(* Logix 5000 project; controller VET 1756-L62 rev 19.52; software revision 19.01; part 27 of 27 *)
(* tags used below, declared in another part *)
   Aux : DINT[40];
   Color_aux : INT[1000];
   ti : Index;
   _Eqp : Equipo[800];
   _Eqp_Cfg : Eqp_Cfg[800];
   _Origen : Origen[40];
   Set_Global : DINT[20];
(* Typlgie, continued *)

ROUTINE SEQ_MOT_1   (* ladder *)
// Parte 1 se seq. equipos
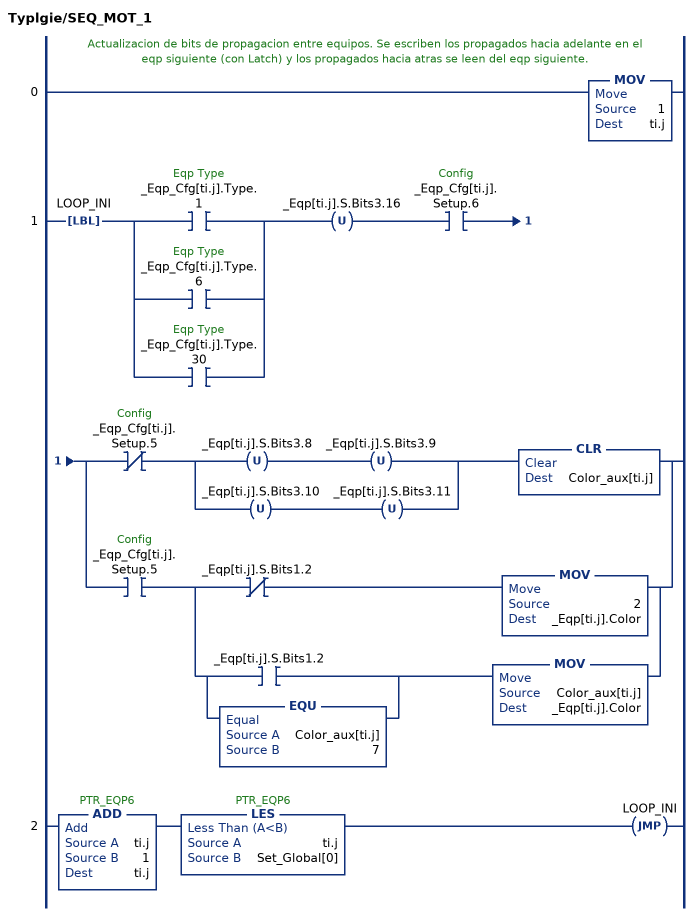
   // Actualizacion de bits de propagacion entre equipos. Se escriben los propagados hacia adelante en el eqp siguiente (con Latch) y los propagados hacia atras se leen del eqp siguiente.
   0: MOV(1,ti.j);
   1: LBL(LOOP_INI)[XIC(_Eqp_Cfg[ti.j].Type.1) ,XIC(_Eqp_Cfg[ti.j].Type.6) ,XIC(_Eqp_Cfg[ti.j].Type.30) ]OTU(_Eqp[ti.j].S.Bits3.16)XIC(_Eqp_Cfg[ti.j].Setup.6)[XIO(_Eqp_Cfg[ti.j].Setup.5) [OTU(_Eqp[ti.j].S.Bits3.8) OTU(_Eqp[ti.j].S.Bits3.9) ,OTU(_Eqp[ti.j].S.Bits3.10) OTU(_Eqp[ti.j].S.Bits3.11) ] CLR(Color_aux[ti.j]) ,XIC(_Eqp_Cfg[ti.j].Setup.5) [XIO(_Eqp[ti.j].S.Bits1.2) MOV(2,_Eqp[ti.j].Color) ,[XIC(_Eqp[ti.j].S.Bits1.2) ,EQU(Color_aux[ti.j],7) ] MOV(Color_aux[ti.j],_Eqp[ti.j].Color) ] ];
   2: ADD(ti.j,1,ti.j)LES(ti.j,Set_Global[0])JMP(LOOP_INI);
END_ROUTINE

ROUTINE SEQ_MOT_2   (* ladder *)
// Parte 2 se seq. equipos
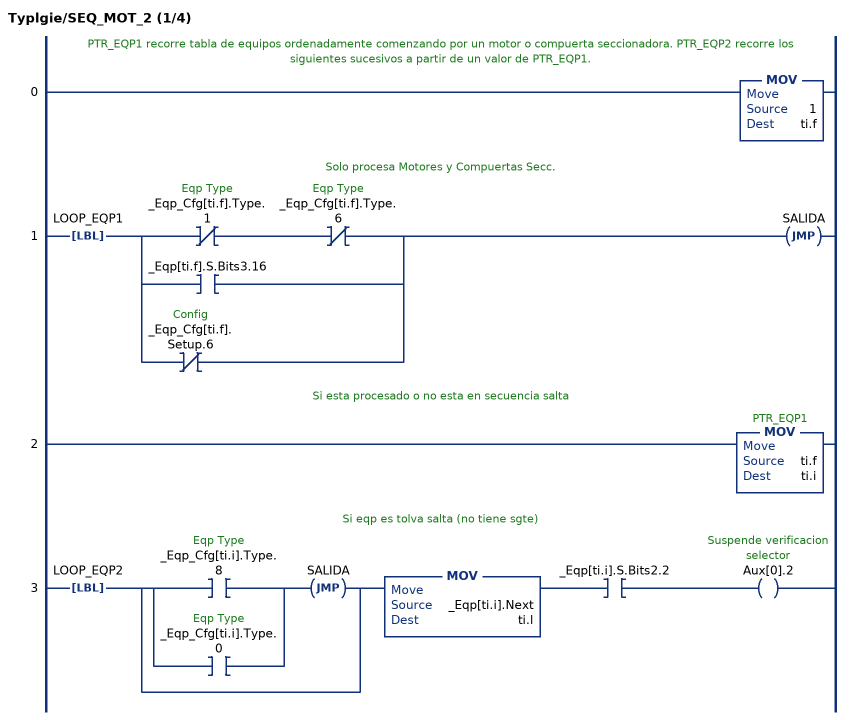
   // PTR_EQP1 recorre tabla de equipos ordenadamente comenzando por un motor o compuerta seccionadora. PTR_EQP2 recorre los siguientes sucesivos a partir de un valor de PTR_EQP1.
   0: MOV(1,ti.f);
   // Solo procesa Motores y Compuertas Secc.
   1: LBL(LOOP_EQP1)[XIO(_Eqp_Cfg[ti.f].Type.1) XIO(_Eqp_Cfg[ti.f].Type.6) ,XIC(_Eqp[ti.f].S.Bits3.16) ,XIO(_Eqp_Cfg[ti.f].Setup.6) ]JMP(SALIDA);
   // Si esta procesado o no esta en secuencia salta
   2: MOV(ti.f,ti.i);
   // Si eqp es tolva salta (no tiene sgte)
   3: LBL(LOOP_EQP2)[[XIC(_Eqp_Cfg[ti.i].Type.8) ,XIC(_Eqp_Cfg[ti.i].Type.0) ] JMP(SALIDA) ,]MOV(_Eqp[ti.i].Next,ti.l)XIC(_Eqp[ti.i].S.Bits2.2)OTE(Aux[0].2);
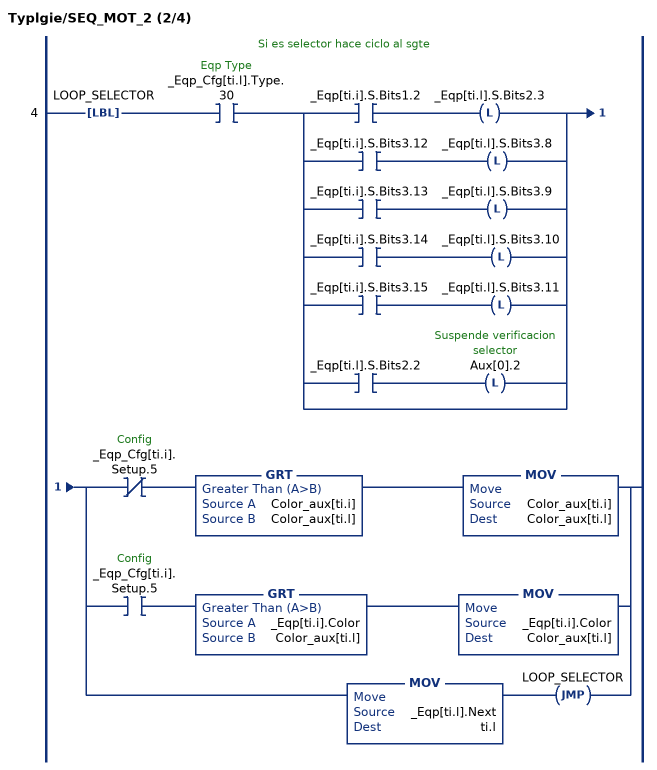
   // Si es selector hace ciclo al sgte
   4: LBL(LOOP_SELECTOR)XIC(_Eqp_Cfg[ti.l].Type.30)[XIC(_Eqp[ti.i].S.Bits1.2) OTL(_Eqp[ti.l].S.Bits2.3) ,XIC(_Eqp[ti.i].S.Bits3.12) OTL(_Eqp[ti.l].S.Bits3.8) ,XIC(_Eqp[ti.i].S.Bits3.13) OTL(_Eqp[ti.l].S.Bits3.9) ,XIC(_Eqp[ti.i].S.Bits3.14) OTL(_Eqp[ti.l].S.Bits3.10) ,XIC(_Eqp[ti.i].S.Bits3.15) OTL(_Eqp[ti.l].S.Bits3.11) ,XIC(_Eqp[ti.l].S.Bits2.2) OTL(Aux[0].2) ,][XIO(_Eqp_Cfg[ti.i].Setup.5) GRT(Color_aux[ti.i],Color_aux[ti.l]) MOV(Color_aux[ti.i],Color_aux[ti.l]) ,XIC(_Eqp_Cfg[ti.i].Setup.5) GRT(_Eqp[ti.i].Color,Color_aux[ti.l]) MOV(_Eqp[ti.i].Color,Color_aux[ti.l]) ,MOV(_Eqp[ti.l].Next,ti.l) JMP(LOOP_SELECTOR) ];
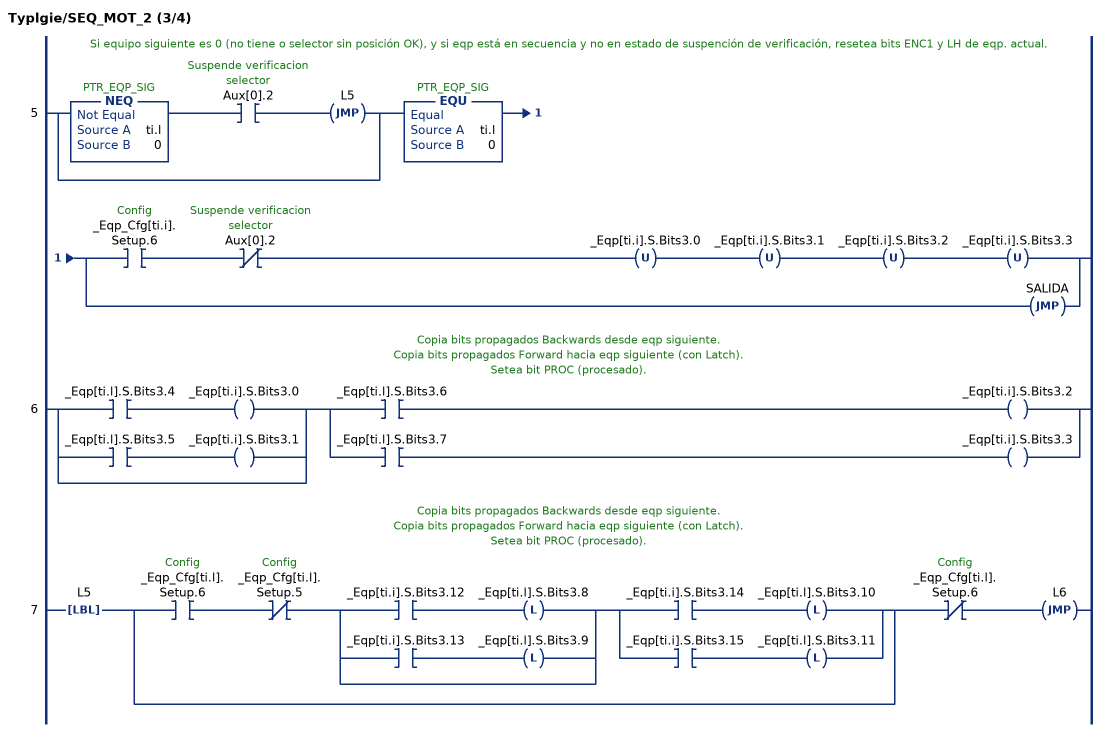
   // Si equipo siguiente es 0 (no tiene o selector sin posición OK), y si eqp está en secuencia y no en estado de suspención de verificación, resetea bits ENC1 y LH de eqp. actual.
   5: [NEQ(ti.l,0) XIC(Aux[0].2) JMP(L5) ,]EQU(ti.l,0)[XIC(_Eqp_Cfg[ti.i].Setup.6) XIO(Aux[0].2) OTU(_Eqp[ti.i].S.Bits3.0) OTU(_Eqp[ti.i].S.Bits3.1) OTU(_Eqp[ti.i].S.Bits3.2) OTU(_Eqp[ti.i].S.Bits3.3) ,JMP(SALIDA) ];
   // Copia bits propagados Backwards desde eqp siguiente.
   // Copia bits propagados Forward hacia eqp siguiente (con Latch).
   // Setea bit PROC (procesado).
   6: [XIC(_Eqp[ti.l].S.Bits3.4) OTE(_Eqp[ti.i].S.Bits3.0) ,XIC(_Eqp[ti.l].S.Bits3.5) OTE(_Eqp[ti.i].S.Bits3.1) ,][XIC(_Eqp[ti.l].S.Bits3.6) OTE(_Eqp[ti.i].S.Bits3.2) ,XIC(_Eqp[ti.l].S.Bits3.7) OTE(_Eqp[ti.i].S.Bits3.3) ];
   // Copia bits propagados Backwards desde eqp siguiente.
   // Copia bits propagados Forward hacia eqp siguiente (con Latch).
   // Setea bit PROC (procesado).
   7: LBL(L5)[XIC(_Eqp_Cfg[ti.l].Setup.6) XIO(_Eqp_Cfg[ti.l].Setup.5) [XIC(_Eqp[ti.i].S.Bits3.12) OTL(_Eqp[ti.l].S.Bits3.8) ,XIC(_Eqp[ti.i].S.Bits3.13) OTL(_Eqp[ti.l].S.Bits3.9) ,] [XIC(_Eqp[ti.i].S.Bits3.14) OTL(_Eqp[ti.l].S.Bits3.10) ,XIC(_Eqp[ti.i].S.Bits3.15) OTL(_Eqp[ti.l].S.Bits3.11) ] ,]XIO(_Eqp_Cfg[ti.l].Setup.6)JMP(L6);
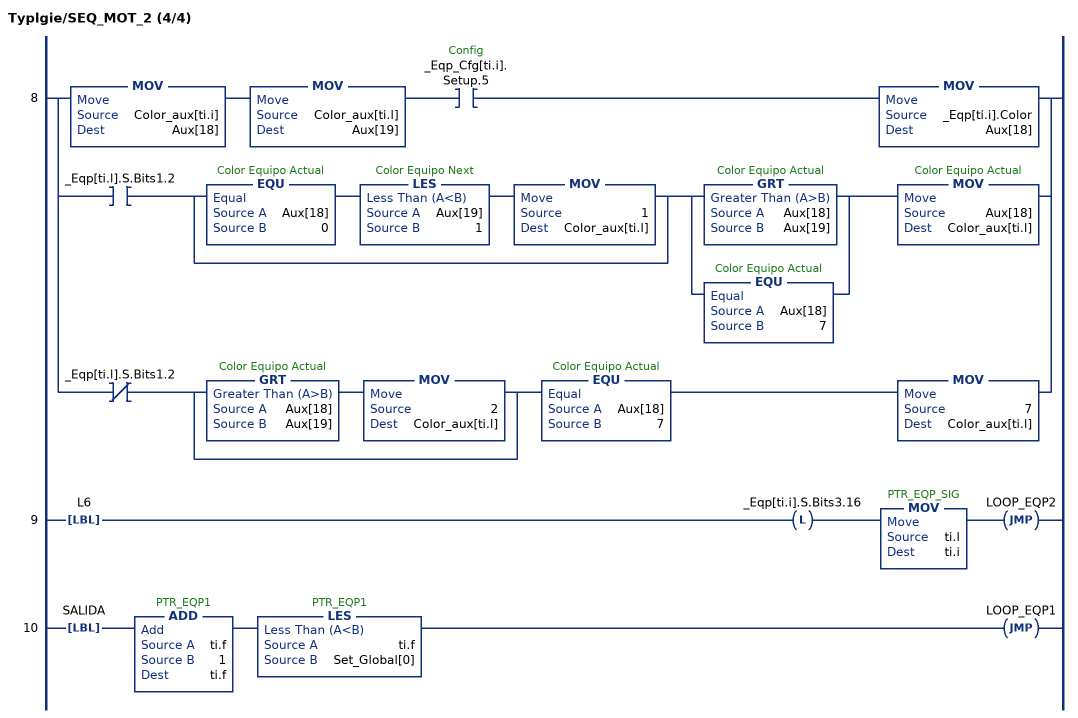
   8: [MOV(Color_aux[ti.i],Aux[18]) MOV(Color_aux[ti.l],Aux[19]) XIC(_Eqp_Cfg[ti.i].Setup.5) MOV(_Eqp[ti.i].Color,Aux[18]) ,XIC(_Eqp[ti.l].S.Bits1.2) [EQU(Aux[18],0) LES(Aux[19],1) MOV(1,Color_aux[ti.l]) ,] [GRT(Aux[18],Aux[19]) ,EQU(Aux[18],7) ] MOV(Aux[18],Color_aux[ti.l]) ,XIO(_Eqp[ti.l].S.Bits1.2) [GRT(Aux[18],Aux[19]) MOV(2,Color_aux[ti.l]) ,] EQU(Aux[18],7) MOV(7,Color_aux[ti.l]) ];
   9: LBL(L6)OTL(_Eqp[ti.i].S.Bits3.16)MOV(ti.l,ti.i)JMP(LOOP_EQP2);
   10: LBL(SALIDA)ADD(ti.f,1,ti.f)LES(ti.f,Set_Global[0])JMP(LOOP_EQP1);
END_ROUTINE

ROUTINE Startup   (* ladder *)
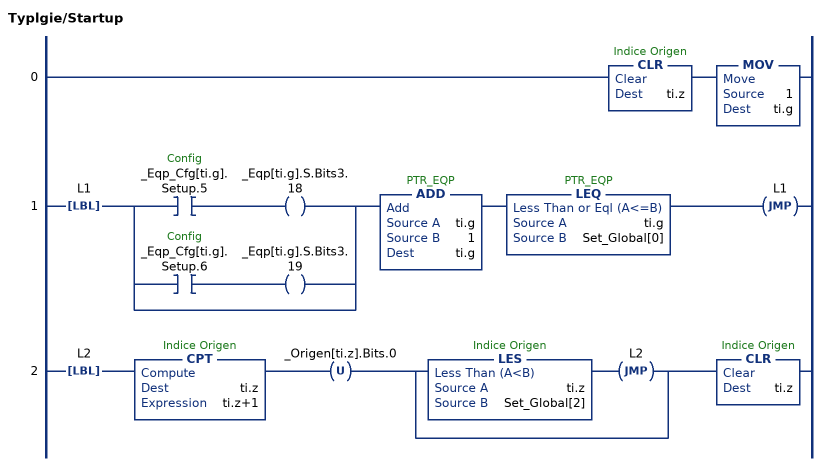
   0: CLR(ti.z)MOV(1,ti.g);
   1: LBL(L1)[XIC(_Eqp_Cfg[ti.g].Setup.5) OTE(_Eqp[ti.g].S.Bits3.18) ,XIC(_Eqp_Cfg[ti.g].Setup.6) OTE(_Eqp[ti.g].S.Bits3.19) ,]ADD(ti.g,1,ti.g)LEQ(ti.g,Set_Global[0])JMP(L1);
   2: LBL(L2)CPT(ti.z,ti.z+1)OTU(_Origen[ti.z].Bits.0)[LES(ti.z,Set_Global[2]) JMP(L2) ,]CLR(ti.z);
END_ROUTINE
END_PROGRAM
